PROGRAM MAIN
VAR
END_VAR

END_PROGRAM

(* stored: Version 1.1.0.1
   POU MAIN: Id {5297f228-285b-46bd-98c4-c531a704c739} *)
